FUNCTION putUdint : BOOL
	VAR_INPUT
		udintVar : UDINT;
	END_VAR
	VAR_IN_OUT
		bufferRef : POINTER TO USINT;
	END_VAR

	memcpy(bufferRef, ADR(udintVar), SIZEOF(UDINT));
	bufferRef := bufferRef + SIZEOF(UDINT);
	putUdint := TRUE;

END_FUNCTION

(* stored: Version 1.1.0.1, ProductVersion 3.1.4024.3
   POU putUdint: Id {ecab3789-ee9c-02bc-3240-0c21f377453e}, SpecialFunc None *)
